// TIA Portal V14 SP1 export
// export: Created 2019-08-14T06:19:05.5821085Z, ExportSetting WithDefaults, WithReadOnly, DisplayName Totally Integrated Automation Portal, DisplayVersion V14 SP1 Update 6, DisplayName TIA Portal Openness, DisplayVersion V14 SP1 Update 6, DisplayName STEP 7 Professional, DisplayVersion V14 SP1 Update 6, DisplayName WinCC Professional, DisplayVersion V14 SP1 Update 6
FUNCTION_BLOCK "554YV_Filter"   // FB2444, LAD
TITLE = Блок управления клапанами очитки фильтра дозатора муки
{ S7_Optimized_Access := 'FALSE' }
VERSION : 0.1
// stored: AutoNumber false, CodeModifiedDate 2019-08-14T06:18:57.2686442Z, CompileDate 2019-08-14T06:18:57.2686441Z, CreationDate 2019-08-14T06:17:58.8399917Z, InterfaceModifiedDate 2019-08-14T06:17:58.8399917Z, IsConsistent true, IsIECCheckEnabled false, IsKnowHowProtected false, ISMultiInstanceCapable true, IsWriteProtected false, LibraryConformanceStatus Warning: The block contains direct access to inputs, outputs, bit memories, indirect access to the registry or indirect access to external memory areas that are unknown at the time of compilation., ModifiedDate 2019-08-14T06:18:57.2686442Z, ParameterModified 2019-08-14T06:17:58.8399917Z, StructureModified 2019-08-14T06:17:58.8399917Z, UDAEnableTagReadback false
   VAR DB_SPECIFIC
      HMI : Struct
         CMD { ExternalVisible := 'False'} : Struct
            Start { ExternalVisible := 'False'} : Bool;   // Старт обрушения в ручном
            Stop { ExternalVisible := 'False'} : Bool;   // Стоп обрушенияи в ручном
            ManCmd_Start { ExternalVisible := 'False'} : Bool;   // Запущено выполнение цикла в ручном режиме
            V2_Disable { ExternalVisible := 'False'} : Bool;   // Клапан 2 выключен
            V3_Disable { ExternalVisible := 'False'} : Bool;   // Клапан 3 выключен
            V4_Disable { ExternalVisible := 'False'} : Bool;   // Клапан 4 выключен
            Manual { ExternalVisible := 'False'} : Bool;   // Ручной режим управления
            FaultReset { ExternalVisible := 'False'} : Bool;   // Сброс ошибок
            CleanTime_priority { ExternalVisible := 'False'} : Bool;
            Spare { ExternalVisible := 'False'} : Bool;
            Spare_1 { ExternalVisible := 'False'} : Bool;
            Spare_2 { ExternalVisible := 'False'} : Bool;
            Spare_3 { ExternalVisible := 'False'} : Bool;
            Spare_4 { ExternalVisible := 'False'} : Bool;
            Spare_5 { ExternalVisible := 'False'} : Bool;
            Spare_6 { ExternalVisible := 'False'} : Bool;
         END_STRUCT;
         DATA : Struct
            StateWord : Word;
            CountDown_Time : Time := T#10s;   // Обратный отсчет цикла очистки / Обратный отсчет цикла обрушения
            CleanTime : Time := T#40s;   // Общее время очистки / Общее время обрушения
            NumberOfCleanings : DInt := 1;   // Количество циклов очистки / Количество циклов обрушения
            Time_Open : Time := T#1s;   // Задание времени работы клапана очистки / Задание времени работы клапана обрушения
            Time_Pause : Time := T#7s;   // Задание времени паузы клапанов очистки / Задание времени паузы клапанов обрушения
            Number_Nozzles : DInt := 4;   // Количество сопел
         END_STRUCT;
      END_STRUCT;
   END_VAR
   VAR
      "844YE" : "Valves_CleanAspirationFilter";
      CycleTimer : TON;
   END_VAR
   VAR DB_SPECIFIC
      Reset_Error : Bool;   // Сброс ошибок / Dumping of errors of the control package
      General_cond_OK : Bool;   // Готовность систем управления / Conditions of permission of operation of the mechanism are not satisfied
      ManCmd_Start : Bool;   // Команда старт обрушения в ручном режиме / Existence of command for rotation of the motor in manual
      ManCmd_Stop : Bool;   // Команда стоп обрушения в ручном режиме / Existence of command for a stop of rotation of the motor in manual
      AutoCmd_Start : Bool;   // Команда старт обрушения в автоматическом режиме / Existence of command for rotation of the motor in the automatic
      AutoCmd_Stop : Bool;   // Команда стоп обрушения в автоматическом режиме / Existence of command for a stop of rotation of the motor in the automatic
      HopperLoad_memo : Bool;
   END_VAR
   VAR_TEMP
      TempBit : Bool;
      Temp_DINT1 : DInt;
      Temp_DINT2 : DInt;
      CycleTime : Time;
   END_VAR
BEGIN

REGION Network 1: Сброс ошибок / СБРОС
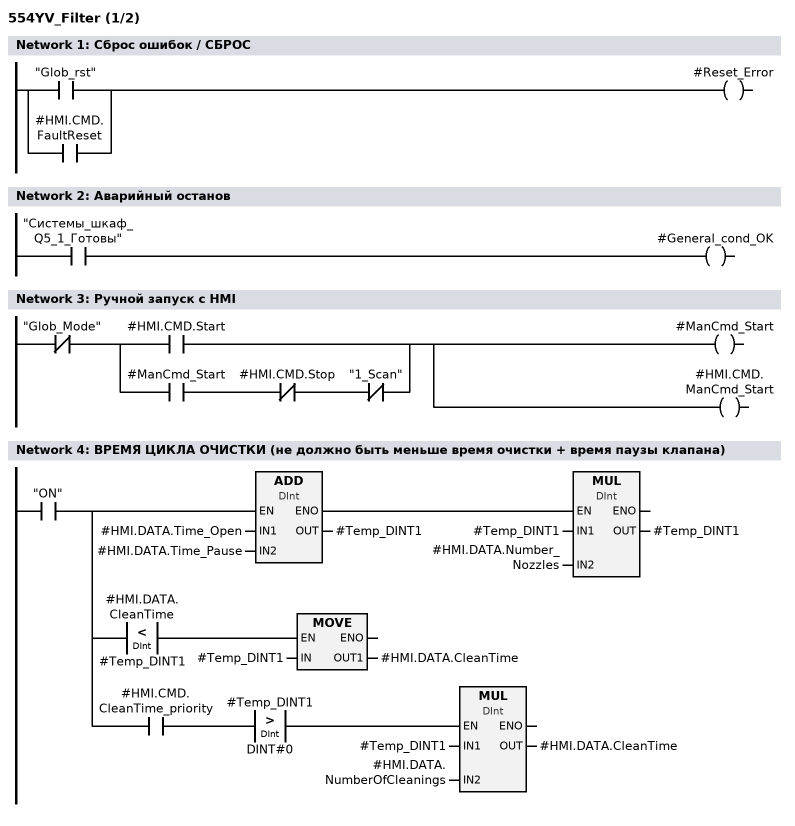
   RUNG wire#powerrail
      Contact( "Glob_rst" )
      wire#w1
      Coil( #Reset_Error )
   END_RUNG
   RUNG wire#powerrail
      Contact( #HMI.CMD.FaultReset )
   END_RUNG wire#w1
   // the same network as SCL:
   #Reset_Error := "Glob_rst" OR #HMI.CMD.FaultReset;
END_REGION

REGION Network 2: Аварийный останов
   RUNG wire#powerrail
      Contact( "Системы_шкаф_Q5_1_Готовы" )
      Coil( #General_cond_OK )
   END_RUNG
   // the same network as SCL:
   #General_cond_OK := "Системы_шкаф_Q5_1_Готовы";
END_REGION

REGION Network 3: Ручной запуск с HMI
   RUNG wire#powerrail
      I_Contact( "Glob_Mode" )
      wire#w1
      Contact( #HMI.CMD.Start )
      wire#w2
      Coil( #ManCmd_Start )
   END_RUNG
   RUNG wire#w1
      Contact( #ManCmd_Start )
      I_Contact( #HMI.CMD.Stop )
      I_Contact( "1_Scan" )
   END_RUNG wire#w2
   RUNG wire#w2
      Coil( #HMI.CMD.ManCmd_Start )
   END_RUNG
   // the same network as SCL:
   #ManCmd_Start := NOT "Glob_Mode" AND (#HMI.CMD.Start OR (#ManCmd_Start AND NOT #HMI.CMD.Stop AND NOT "1_Scan"));
   #HMI.CMD.ManCmd_Start := #ManCmd_Start;
END_REGION

REGION Network 4: ВРЕМЯ ЦИКЛА ОЧИСТКИ (не должно быть меньше время очистки + время паузы клапана)
   RUNG wire#powerrail
      Contact( "ON" )
      wire#w1
      { S7_Templates := "SrcType := DInt"; S7_GenerateENO := "TRUE" } Add(in1 := #HMI.DATA.Time_Open, in2 := #HMI.DATA.Time_Pause, out => #Temp_DINT1)
      { S7_Templates := "SrcType := DInt"; S7_GenerateENO := "TRUE" } Mul(in1 := #Temp_DINT1, in2 := #HMI.DATA.Number_Nozzles, out => #Temp_DINT1)
   END_RUNG
   RUNG wire#w1
      { S7_Templates := "SrcType := DInt" } LT_Contact(in1 := #HMI.DATA.CleanTime, in2 := #Temp_DINT1)
      { S7_GenerateENO := "TRUE" } Move(in := #Temp_DINT1, out1 => #HMI.DATA.CleanTime)
   END_RUNG
   RUNG wire#w1
      Contact( #HMI.CMD.CleanTime_priority )
      { S7_Templates := "SrcType := DInt" } GT_Contact(in1 := #Temp_DINT1, in2 := DINT#0)
      { S7_Templates := "SrcType := DInt"; S7_GenerateENO := "TRUE" } Mul(in1 := #Temp_DINT1, in2 := #HMI.DATA.NumberOfCleanings, out => #HMI.DATA.CleanTime)
   END_RUNG
   // the same network as SCL:
   // ENO of a box is taken as its EN; it also drops when the box reports an error
   IF "ON" THEN
       #Temp_DINT1 := #HMI.DATA.Time_Open + #HMI.DATA.Time_Pause;
       #Temp_DINT1 := #Temp_DINT1 * #HMI.DATA.Number_Nozzles;
   END_IF;
   IF "ON" AND (#HMI.DATA.CleanTime < #Temp_DINT1) THEN #HMI.DATA.CleanTime := #Temp_DINT1; END_IF;
   IF "ON" AND #HMI.CMD.CleanTime_priority AND (#Temp_DINT1 > DINT#0) THEN
       #HMI.DATA.CleanTime := #Temp_DINT1 * #HMI.DATA.NumberOfCleanings;
   END_IF;
END_REGION

REGION Network 5: ЗАПУСК ЦИКЛА
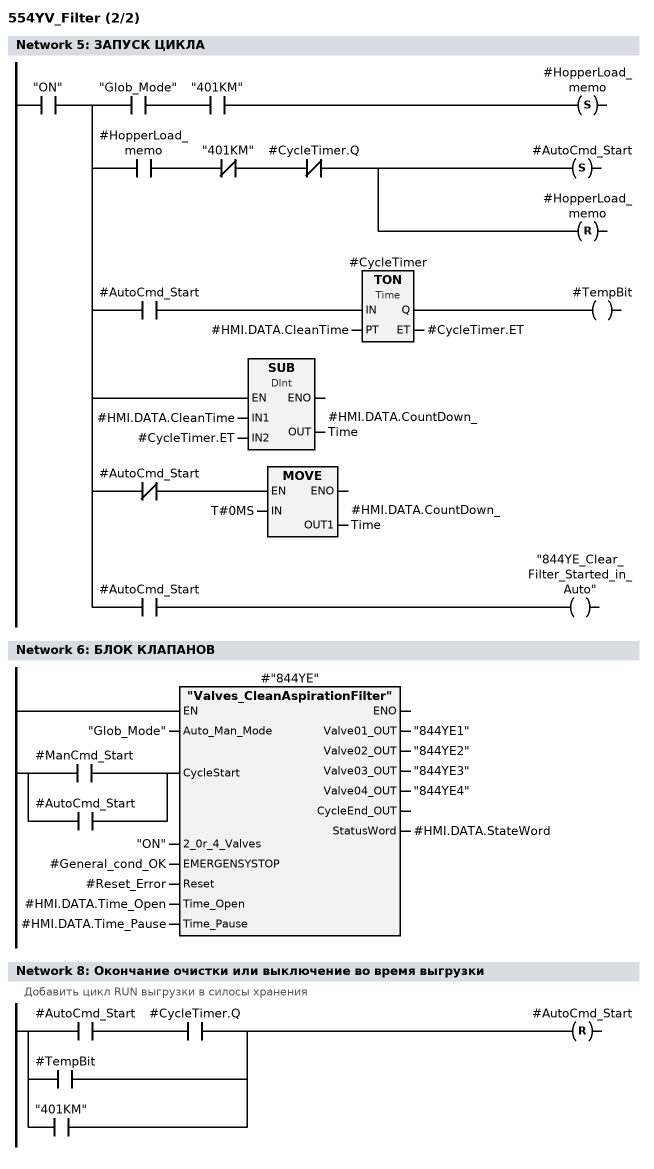
   RUNG wire#powerrail
      Contact( "ON" )
      wire#w1
      Contact( "Glob_Mode" )
      Contact( "401KM" )
      S_Coil( #HopperLoad_memo )
   END_RUNG
   RUNG wire#w1
      Contact( #HopperLoad_memo )
      I_Contact( "401KM" )
      I_Contact( #CycleTimer.Q )
      wire#w2
      S_Coil( #AutoCmd_Start )
   END_RUNG
   RUNG wire#w2
      R_Coil( #HopperLoad_memo )
   END_RUNG
   RUNG wire#w1
      Contact( #AutoCmd_Start )
      { S7_Templates := "time_type := Time" } #CycleTimer.TON(pt := #HMI.DATA.CleanTime, et => #CycleTimer.ET)
      Coil( #TempBit )
   END_RUNG
   RUNG wire#w1
      { S7_Templates := "SrcType := DInt"; S7_GenerateENO := "TRUE" } Sub(in1 := #HMI.DATA.CleanTime, in2 := #CycleTimer.ET, out => #HMI.DATA.CountDown_Time)
   END_RUNG
   RUNG wire#w1
      I_Contact( #AutoCmd_Start )
      { S7_GenerateENO := "TRUE" } Move(in := T#0MS, out1 => #HMI.DATA.CountDown_Time)
   END_RUNG
   RUNG wire#w1
      Contact( #AutoCmd_Start )
      Coil( "844YE_Clear_Filter_Started_in_Auto" )
   END_RUNG
   // the same network as SCL:
   IF "ON" AND "Glob_Mode" AND "401KM" THEN #HopperLoad_memo := TRUE; END_IF;
   IF "ON" AND #HopperLoad_memo AND NOT "401KM" AND NOT #CycleTimer.Q THEN
       #AutoCmd_Start := TRUE;
       #HopperLoad_memo := FALSE;
   END_IF;
   #CycleTimer.TON(IN := "ON" AND #AutoCmd_Start, PT := #HMI.DATA.CleanTime, ET => #CycleTimer.ET);
   #TempBit := #CycleTimer.Q;
   IF "ON" THEN #HMI.DATA.CountDown_Time := #HMI.DATA.CleanTime - #CycleTimer.ET; END_IF;
   IF "ON" AND NOT #AutoCmd_Start THEN #HMI.DATA.CountDown_Time := T#0MS; END_IF;
   "844YE_Clear_Filter_Started_in_Auto" := "ON" AND #AutoCmd_Start;
END_REGION

REGION Network 6: БЛОК КЛАПАНОВ
   RUNG wire#powerrail
      #"844YE"(CycleStart := wire#w1, Auto_Man_Mode := "Glob_Mode", "2_0r_4_Valves" := "ON", EMERGENSYSTOP := #General_cond_OK, Reset := #Reset_Error, Time_Open := #HMI.DATA.Time_Open, Time_Pause := #HMI.DATA.Time_Pause, Valve01_OUT => "844YE1", Valve02_OUT => "844YE2", Valve03_OUT => "844YE3", Valve04_OUT => "844YE4", CycleEnd_OUT =>, StatusWord => #HMI.DATA.StateWord)
   END_RUNG
   RUNG wire#powerrail
      Contact( #ManCmd_Start )
   END_RUNG wire#w1
   RUNG wire#powerrail
      Contact( #AutoCmd_Start )
   END_RUNG wire#w1
   // the same network as SCL:
   #"844YE"(Auto_Man_Mode := "Glob_Mode",   // "Valves_CleanAspirationFilter"
            CycleStart := #ManCmd_Start OR #AutoCmd_Start,
            "2_0r_4_Valves" := "ON",
            EMERGENSYSTOP := #General_cond_OK,
            Reset := #Reset_Error,
            Time_Open := #HMI.DATA.Time_Open,
            Time_Pause := #HMI.DATA.Time_Pause,
            Valve01_OUT => "844YE1",
            Valve02_OUT => "844YE2",
            Valve03_OUT => "844YE3",
            Valve04_OUT => "844YE4",
            StatusWord => #HMI.DATA.StateWord);
END_REGION

REGION Network 7: END
END_REGION

REGION Network 8: Окончание очистки или выключение во время выгрузки
   // Добавить цикл RUN выгрузки в силосы хранения
   RUNG wire#powerrail
      Contact( #AutoCmd_Start )
      Contact( #CycleTimer.Q )
      wire#w1
      R_Coil( #AutoCmd_Start )
   END_RUNG
   RUNG wire#powerrail
      Contact( #TempBit )
   END_RUNG wire#w1
   RUNG wire#powerrail
      Contact( "401KM" )
   END_RUNG wire#w1
   // the same network as SCL:
   IF (#AutoCmd_Start AND #CycleTimer.Q) OR #TempBit OR "401KM" THEN #AutoCmd_Start := FALSE; END_IF;
END_REGION
END_FUNCTION_BLOCK
